{attribute 'qualified_only'}
{attribute 'strict'}
TYPE E_PTC_TX_Command :
(
	HV_ON := 16#04,
	HV_OFF := 16#0B,
	PreCharge_Reset := 16#03,
	Clear_PreCharge_Failure := 16#01
)BYTE;
END_TYPE

(* stored: Version 1.1.0.1
   DUT E_PTC_TX_Command: Id {afee7328-5fc0-40c4-8b32-845ce91942a8} *)
